// TwinCAT 3 PLC project PlcTcProberTests
// ProgramVersion: 3.1.4023.0
// libraries:
//   Tc2_Standard, * (Beckhoff Automation GmbH)
//   Tc2_System, * (Beckhoff Automation GmbH)
//   Tc3_Module, * (Beckhoff Automation GmbH)
// project tree:
//   GVLs/ Tests.TcGVL
//   / PlcTask.TcTTO (not stored)
//   POUs/ MAIN.TcPOU
//   Runners/ fbBasicRunnerTests.TcPOU (not stored), fbRecorderRunnerTests.TcPOU, stRecorder.TcDUT (not stored)
//   Runners/TestStructs/nestedInheritance/ fbInheritanceLevel_1.TcPOU (not stored), fbInheritanceLevel_2.TcPOU (not stored), fbInheritanceLevel_3.TcPOU (not stored), fbInheritanceLevel_4.TcPOU (not stored), fbInheritanceLevel_5.TcPOU (not stored), fbRootLevelStruct.TcPOU (not stored)
//   Runners/TestStructs/ stAllTypes.TcDUT (not stored)
// real-time tasks:
//   TASK PlcTask: cycle T#10ms, priority 20, ADS port 350

// ---- GVLs/Tests.TcGVL
{attribute 'qualified_only'}
VAR_GLOBAL
	_basicRunnerTests : fbBasicRunnerTests;
END_VAR

// ---- POUs/MAIN.TcPOU
PROGRAM MAIN
VAR
END_VAR

END_PROGRAM

// ---- Runners/fbRecorderRunnerTests.TcPOU
FUNCTION_BLOCK fbRecorderRunnerTests
VAR
    _recorder : stRecorder; 	
END_VAR

{attribute 'TcRpcEnable'}
METHOD ResetCounter : UINT
_recorder.counter := 0;
END_METHOD

{attribute 'TcRpcEnable'}
METHOD RunWithRecorder : UINT
_recorder.counter := _recorder.counter + 1;
END_METHOD

END_FUNCTION_BLOCK
